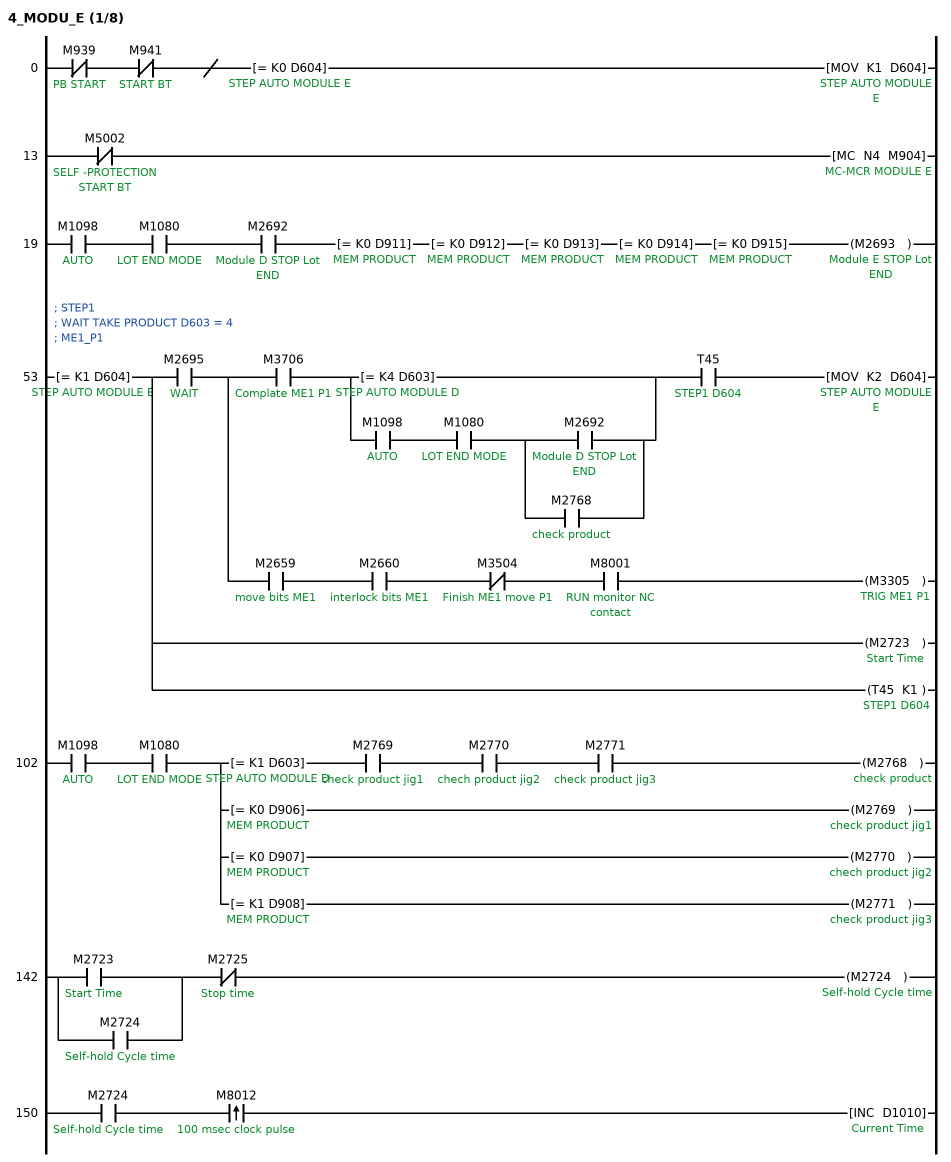
[picture p48: ladder of 4_MODU_E, rungs at steps 0 to 150]
0     LDI     M939  ; PB START
      ANI     M941  ; START BT
      INV
      AND=    K0 D604  ; STEP AUTO MODULE E
      MOV     K1 D604
13    LDI     M5002  ; SELF -PROTECTION START BT
      MC      N4 M904  ; MC-MCR MODULE E
19    LD      M1098  ; AUTO
      AND     M1080  ; LOT END MODE
      AND     M2692  ; Module D STOP Lot END
      AND=    K0 D911  ; MEM PRODUCT
      AND=    K0 D912  ; MEM PRODUCT
      AND=    K0 D913  ; MEM PRODUCT
      AND=    K0 D914  ; MEM PRODUCT
      AND=    K0 D915  ; MEM PRODUCT
      OUT     M2693  ; Module E STOP Lot END
; STEP1
; WAIT TAKE PRODUCT D603 = 4
; ME1_P1
53    LD=     K1 D604  ; STEP AUTO MODULE E
      MPS
      AND     M2695  ; WAIT
      MPS
      AND     M3706  ; Complate ME1 P1
      LD=     K4 D603  ; STEP AUTO MODULE D
      LD      M1098  ; AUTO
      AND     M1080  ; LOT END MODE
      LD      M2692  ; Module D STOP Lot END
      OR      M2768  ; check product
      ANB
      ORB
      ANB
      AND     T45  ; STEP1 D604
      MOV     K2 D604
      MPP
      AND     M2659  ; move bits ME1
      AND     M2660  ; interlock bits ME1
      ANI     M3504  ; Finish ME1 move P1
      AND     M8001  ; RUN monitor NC contact
      OUT     M3305  ; TRIG ME1 P1
        [note] TRIG ME1 P1
      MPP
      OUT     M2723  ; Start Time
      OUT     T45 K1  ; STEP1 D604
102   LD      M1098  ; AUTO
      AND     M1080  ; LOT END MODE
      MPS
      AND=    K1 D603  ; STEP AUTO MODULE D
      AND     M2769  ; check product jig1
      AND     M2770  ; chech product jig2
      AND     M2771  ; check product jig3
      OUT     M2768  ; check product
      MRD
      AND=    K0 D906  ; MEM PRODUCT
      OUT     M2769  ; check product jig1
      MRD
      AND=    K0 D907  ; MEM PRODUCT
      OUT     M2770  ; chech product jig2
      MPP
      AND=    K1 D908  ; MEM PRODUCT
      OUT     M2771  ; check product jig3
142   LD      M2723  ; Start Time
      OR      M2724  ; Self-hold Cycle time
      ANI     M2725  ; Stop time
      OUT     M2724  ; Self-hold Cycle time
150   LD      M2724  ; Self-hold Cycle time
      ANDP    M8012  ; 100 msec clock pulse
      INC     D1010  ; Current Time
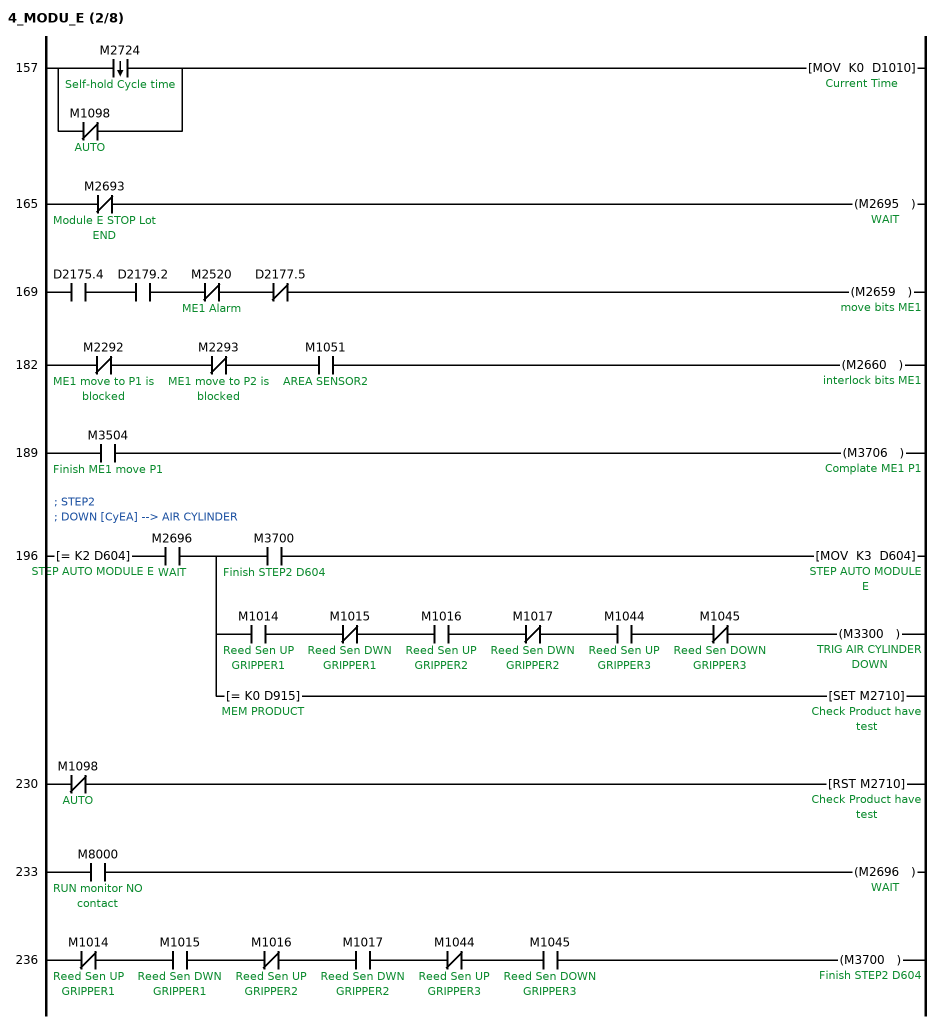
157   LDF     M2724  ; Self-hold Cycle time
      ORI     M1098  ; AUTO
      MOV     K0 D1010
165   LDI     M2693  ; Module E STOP Lot END
      OUT     M2695  ; WAIT
169   LD      D2175.4
      AND     D2179.2
      ANI     M2520  ; ME1 Alarm
      ANI     D2177.5
      OUT     M2659  ; move bits ME1
182   LDI     M2292  ; ME1 move to P1 is blocked
      ANI     M2293  ; ME1 move to P2 is blocked
      AND     M1051  ; AREA SENSOR2
      OUT     M2660  ; interlock bits ME1
189   LD      M3504  ; Finish ME1 move P1
      OUT     M3706  ; Complate ME1 P1
; STEP2
; DOWN [CyEA] --> AIR CYLINDER
196   LD=     K2 D604  ; STEP AUTO MODULE E
      AND     M2696  ; WAIT
      MPS
      AND     M3700  ; Finish STEP2 D604
      MOV     K3 D604
      MRD
      AND     M1014  ; Reed Sen UP GRIPPER1
      ANI     M1015  ; Reed Sen DWN GRIPPER1
      AND     M1016  ; Reed Sen UP GRIPPER2
      ANI     M1017  ; Reed Sen DWN GRIPPER2
      AND     M1044  ; Reed Sen UP GRIPPER3
      ANI     M1045  ; Reed Sen DOWN GRIPPER3
      OUT     M3300  ; TRIG AIR CYLINDER DOWN
        [note] TRIG AIR CYLINDER DOWN
      MPP
      AND=    K0 D915  ; MEM PRODUCT
      SET     M2710  ; Check Product have test
230   LDI     M1098  ; AUTO
      RST     M2710  ; Check Product have test
233   LD      M8000  ; RUN monitor NO contact
      OUT     M2696  ; WAIT
236   LDI     M1014  ; Reed Sen UP GRIPPER1
      AND     M1015  ; Reed Sen DWN GRIPPER1
      ANI     M1016  ; Reed Sen UP GRIPPER2
      AND     M1017  ; Reed Sen DWN GRIPPER2
      ANI     M1044  ; Reed Sen UP GRIPPER3
      AND     M1045  ; Reed Sen DOWN GRIPPER3
      OUT     M3700  ; Finish STEP2 D604
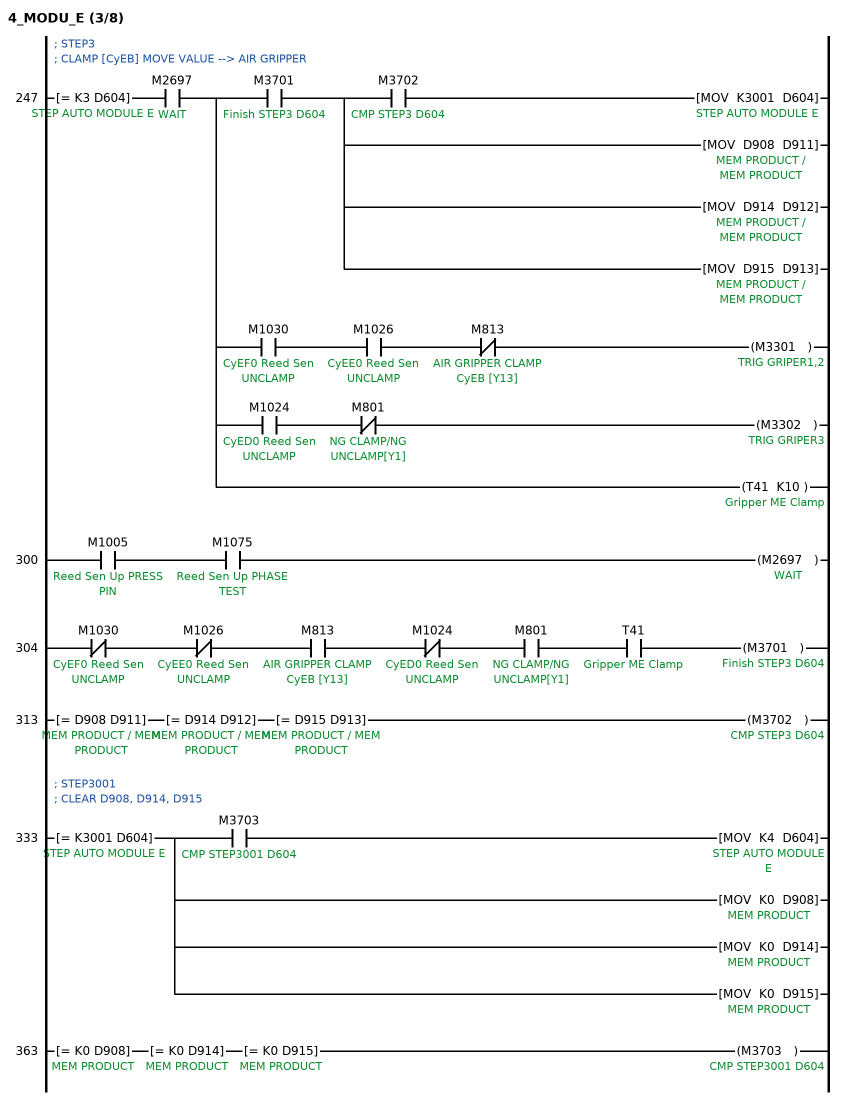
; STEP3
; CLAMP [CyEB] MOVE VALUE --> AIR GRIPPER
247   LD=     K3 D604  ; STEP AUTO MODULE E
      AND     M2697  ; WAIT
      MPS
      AND     M3701  ; Finish STEP3 D604
      MPS
      AND     M3702  ; CMP STEP3 D604
      MOV     K3001 D604
      MPP
      MOV     D908 D911
      MOV     D914 D912
      MOV     D915 D913
      MRD
      AND     M1030  ; CyEF0 Reed Sen UNCLAMP
      AND     M1026  ; CyEE0 Reed Sen UNCLAMP
      ANI     M813  ; AIR GRIPPER CLAMP CyEB [Y13]
      OUT     M3301  ; TRIG GRIPER1,2
        [note] TRIG GRIPER1,2
      MRD
      AND     M1024  ; CyED0 Reed Sen UNCLAMP
      ANI     M801  ; NG CLAMP/NG UNCLAMP[Y1]
      OUT     M3302  ; TRIG GRIPER3
        [note] TRIG GRIPER3
      MPP
      OUT     T41 K10  ; Gripper ME Clamp
300   LD      M1005  ; Reed Sen Up PRESS PIN
      AND     M1075  ; Reed Sen Up PHASE TEST
      OUT     M2697  ; WAIT
304   LDI     M1030  ; CyEF0 Reed Sen UNCLAMP
      ANI     M1026  ; CyEE0 Reed Sen UNCLAMP
      AND     M813  ; AIR GRIPPER CLAMP CyEB [Y13]
      ANI     M1024  ; CyED0 Reed Sen UNCLAMP
      AND     M801  ; NG CLAMP/NG UNCLAMP[Y1]
      AND     T41  ; Gripper ME Clamp
      OUT     M3701  ; Finish STEP3 D604
313   LD=     D908 D911  ; MEM PRODUCT / MEM PRODUCT
      AND=    D914 D912  ; MEM PRODUCT / MEM PRODUCT
      AND=    D915 D913  ; MEM PRODUCT / MEM PRODUCT
      OUT     M3702  ; CMP STEP3 D604
; STEP3001
; CLEAR D908, D914, D915
333   LD=     K3001 D604  ; STEP AUTO MODULE E
      MPS
      AND     M3703  ; CMP STEP3001 D604
      MOV     K4 D604
      MPP
      MOV     K0 D908
      MOV     K0 D914
      MOV     K0 D915
363   LD=     K0 D908  ; MEM PRODUCT
      AND=    K0 D914  ; MEM PRODUCT
      AND=    K0 D915  ; MEM PRODUCT
      OUT     M3703  ; CMP STEP3001 D604
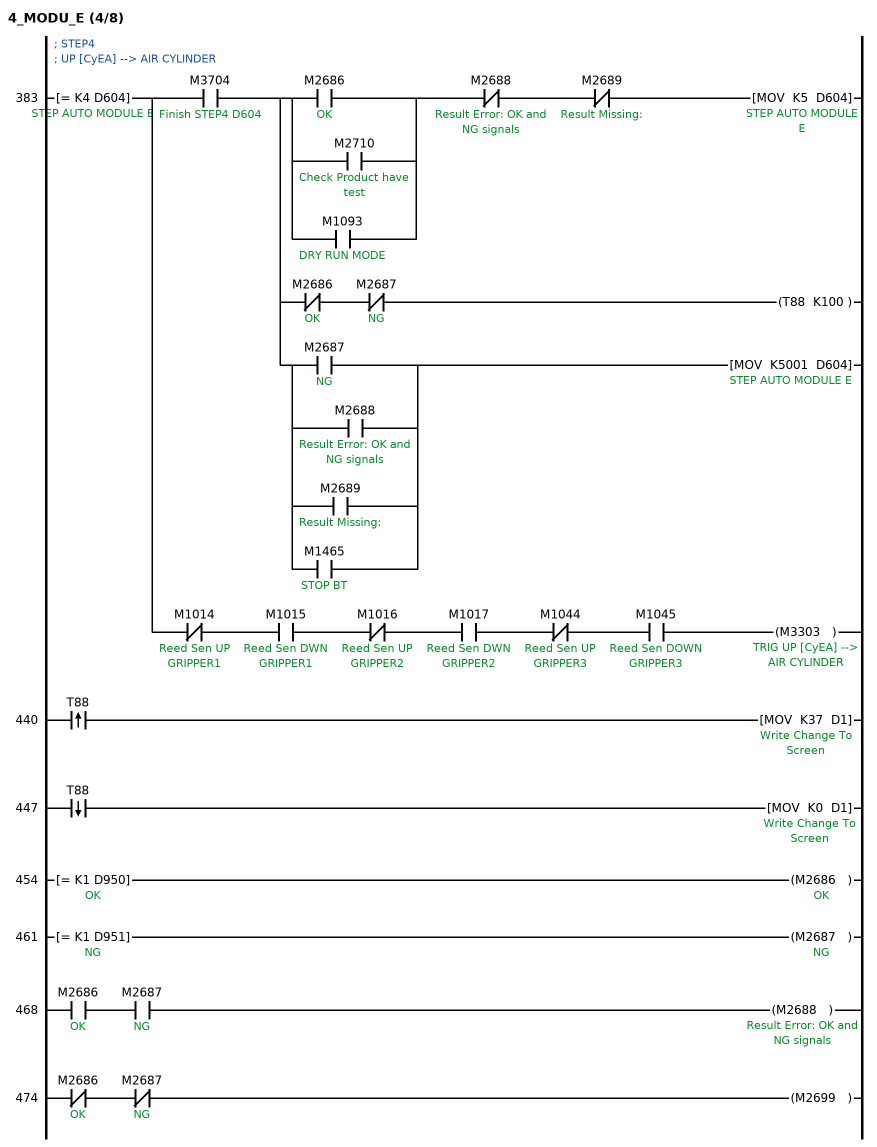
; STEP4
; UP [CyEA] --> AIR CYLINDER
383   LD=     K4 D604  ; STEP AUTO MODULE E
      MPS
      AND     M3704  ; Finish STEP4 D604
      MPS
      LD      M2686  ; OK
      OR      M2710  ; Check Product have test
      OR      M1093  ; DRY RUN MODE
      ANB
      ANI     M2688  ; Result Error: OK and NG signals
      ANI     M2689  ; Result Missing:
      MOV     K5 D604
      MRD
      ANI     M2686  ; OK
      ANI     M2687  ; NG
      OUT     T88 K100
      MPP
      LD      M2687  ; NG
      OR      M2688  ; Result Error: OK and NG signals
      OR      M2689  ; Result Missing:
      OR      M1465  ; STOP BT
      ANB
      MOV     K5001 D604
      MPP
      ANI     M1014  ; Reed Sen UP GRIPPER1
      AND     M1015  ; Reed Sen DWN GRIPPER1
      ANI     M1016  ; Reed Sen UP GRIPPER2
      AND     M1017  ; Reed Sen DWN GRIPPER2
      ANI     M1044  ; Reed Sen UP GRIPPER3
      AND     M1045  ; Reed Sen DOWN GRIPPER3
      OUT     M3303  ; TRIG UP [CyEA] --> AIR CYLINDER
        [note] TRIG UP AIR CYLINDER
440   LDP     T88
      MOV     K37 D1  ; Write Change To Screen
447   LDF     T88
      MOV     K0 D1
454   LD=     K1 D950  ; OK
      OUT     M2686  ; OK
461   LD=     K1 D951  ; NG
      OUT     M2687  ; NG
468   LD      M2686  ; OK
      AND     M2687  ; NG
      OUT     M2688  ; Result Error: OK and NG signals
474   LDI     M2686  ; OK
      ANI     M2687  ; NG
      OUT     M2699
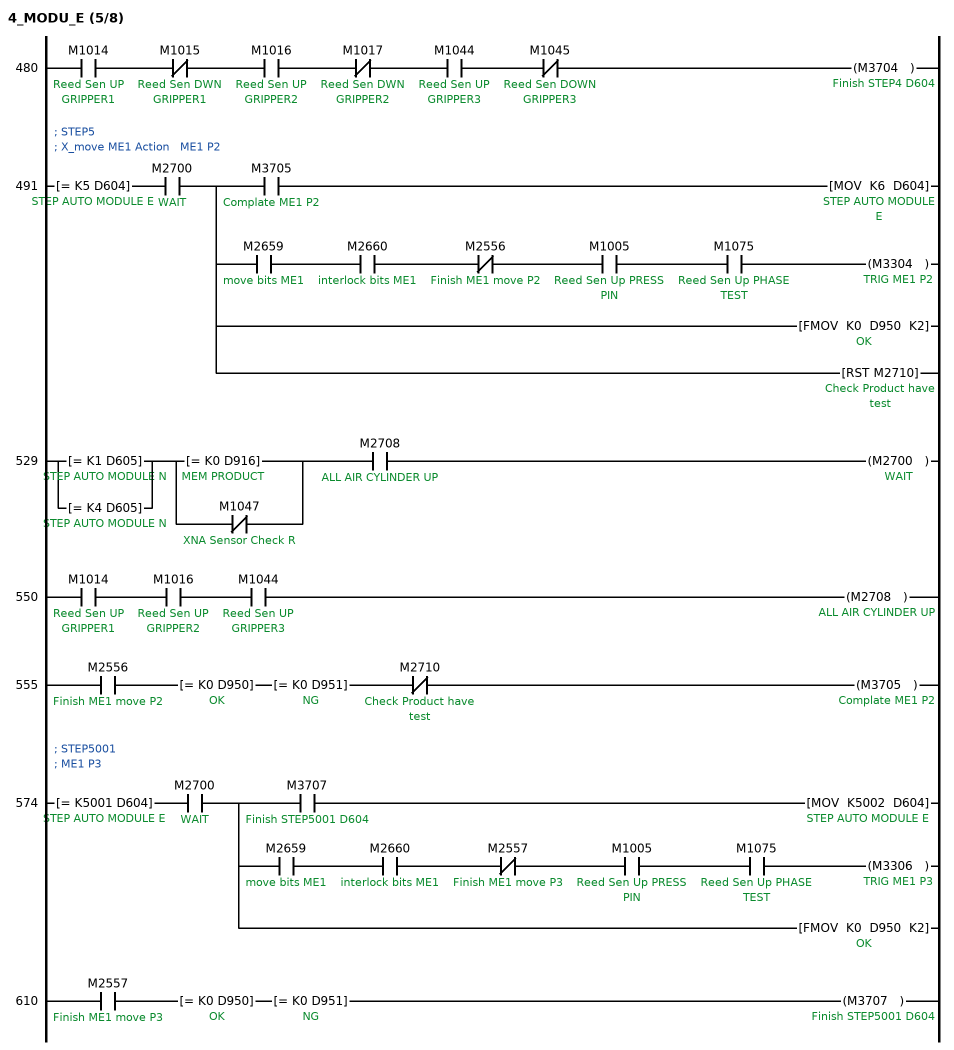
480   LD      M1014  ; Reed Sen UP GRIPPER1
      ANI     M1015  ; Reed Sen DWN GRIPPER1
      AND     M1016  ; Reed Sen UP GRIPPER2
      ANI     M1017  ; Reed Sen DWN GRIPPER2
      AND     M1044  ; Reed Sen UP GRIPPER3
      ANI     M1045  ; Reed Sen DOWN GRIPPER3
      OUT     M3704  ; Finish STEP4 D604
; STEP5
; X_move ME1 Action   ME1 P2
491   LD=     K5 D604  ; STEP AUTO MODULE E
      AND     M2700  ; WAIT
      MPS
      AND     M3705  ; Complate ME1 P2
      MOV     K6 D604
      MRD
      AND     M2659  ; move bits ME1
      AND     M2660  ; interlock bits ME1
      ANI     M2556  ; Finish ME1 move P2
      AND     M1005  ; Reed Sen Up PRESS PIN
      AND     M1075  ; Reed Sen Up PHASE TEST
      OUT     M3304  ; TRIG ME1 P2
        [note] TRIG ME1 P2
      MPP
      FMOV    K0 D950 K2
      RST     M2710  ; Check Product have test
529   LD=     K1 D605  ; STEP AUTO MODULE N
      OR=     K4 D605  ; STEP AUTO MODULE N
      LD=     K0 D916  ; MEM PRODUCT
      ORI     M1047  ; XNA Sensor Check R
      ANB
      AND     M2708  ; ALL AIR CYLINDER UP
      OUT     M2700  ; WAIT
550   LD      M1014  ; Reed Sen UP GRIPPER1
      AND     M1016  ; Reed Sen UP GRIPPER2
      AND     M1044  ; Reed Sen UP GRIPPER3
      OUT     M2708  ; ALL AIR CYLINDER UP
555   LD      M2556  ; Finish ME1 move P2
      AND=    K0 D950  ; OK
      AND=    K0 D951  ; NG
      ANI     M2710  ; Check Product have test
      OUT     M3705  ; Complate ME1 P2
; STEP5001
; ME1 P3
574   LD=     K5001 D604  ; STEP AUTO MODULE E
      AND     M2700  ; WAIT
      MPS
      AND     M3707  ; Finish STEP5001 D604
      MOV     K5002 D604
      MRD
      AND     M2659  ; move bits ME1
      AND     M2660  ; interlock bits ME1
      ANI     M2557  ; Finish ME1 move P3
      AND     M1005  ; Reed Sen Up PRESS PIN
      AND     M1075  ; Reed Sen Up PHASE TEST
      OUT     M3306  ; TRIG ME1 P3
        [note] TRIG ME1 P3
      MPP
      FMOV    K0 D950 K2
610   LD      M2557  ; Finish ME1 move P3
      AND=    K0 D950  ; OK
      AND=    K0 D951  ; NG
      OUT     M3707  ; Finish STEP5001 D604
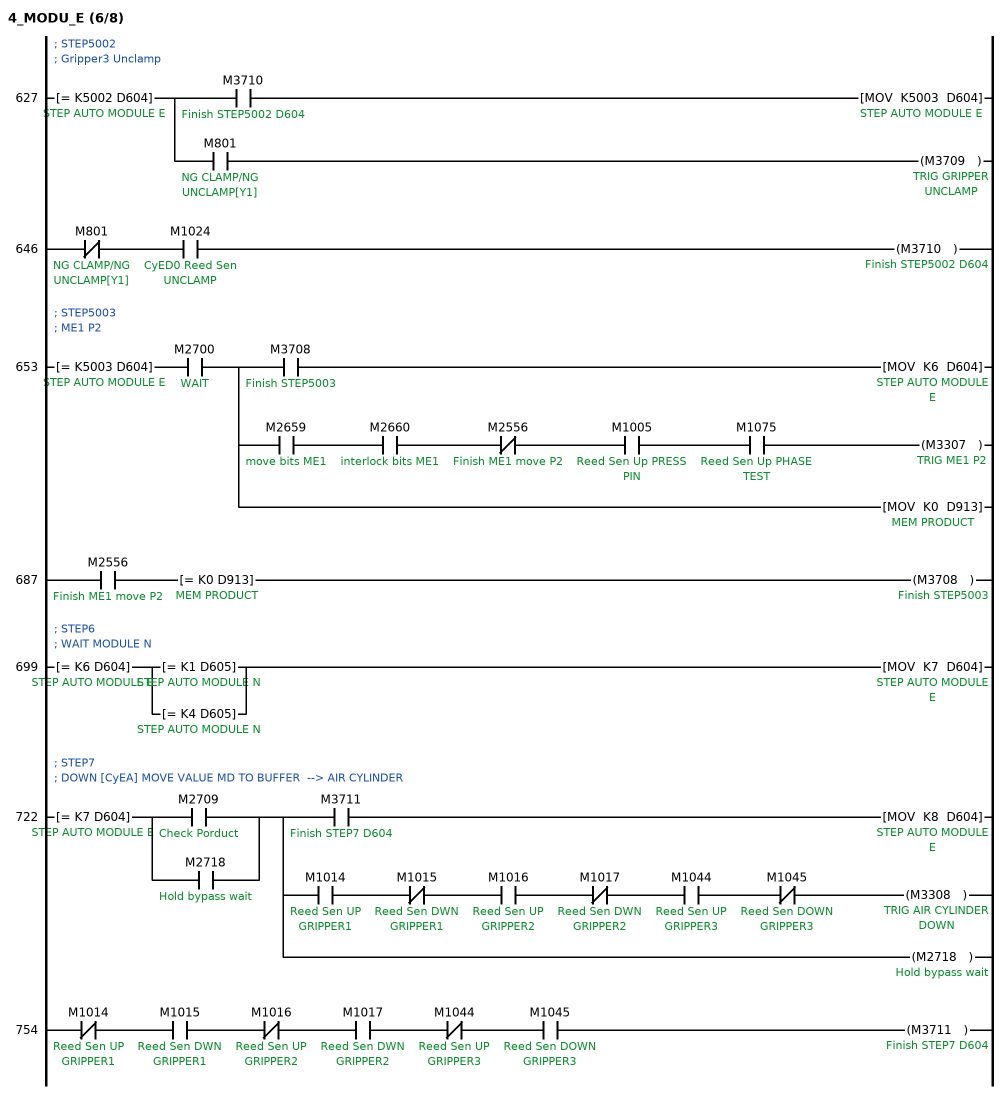
; STEP5002
; Gripper3 Unclamp
627   LD=     K5002 D604  ; STEP AUTO MODULE E
      MPS
      AND     M3710  ; Finish STEP5002 D604
      MOV     K5003 D604
      MPP
      AND     M801  ; NG CLAMP/NG UNCLAMP[Y1]
      OUT     M3709  ; TRIG GRIPPER UNCLAMP
646   LDI     M801  ; NG CLAMP/NG UNCLAMP[Y1]
      AND     M1024  ; CyED0 Reed Sen UNCLAMP
      OUT     M3710  ; Finish STEP5002 D604
; STEP5003
; ME1 P2
653   LD=     K5003 D604  ; STEP AUTO MODULE E
      AND     M2700  ; WAIT
      MPS
      AND     M3708  ; Finish STEP5003
      MOV     K6 D604
      MRD
      AND     M2659  ; move bits ME1
      AND     M2660  ; interlock bits ME1
      ANI     M2556  ; Finish ME1 move P2
      AND     M1005  ; Reed Sen Up PRESS PIN
      AND     M1075  ; Reed Sen Up PHASE TEST
      OUT     M3307  ; TRIG ME1 P2
        [note] TRIG ME1 P2
      MPP
      MOV     K0 D913
687   LD      M2556  ; Finish ME1 move P2
      AND=    K0 D913  ; MEM PRODUCT
      OUT     M3708  ; Finish STEP5003
; STEP6
; WAIT MODULE N
699   LD=     K6 D604  ; STEP AUTO MODULE E
      LD=     K1 D605  ; STEP AUTO MODULE N
      OR=     K4 D605  ; STEP AUTO MODULE N
      ANB
      MOV     K7 D604
; STEP7
; DOWN [CyEA] MOVE VALUE MD TO BUFFER  --> AIR CYLINDER
722   LD=     K7 D604  ; STEP AUTO MODULE E
      LD      M2709  ; Check Porduct
      OR      M2718  ; Hold bypass wait
      ANB
      MPS
      AND     M3711  ; Finish STEP7 D604
      MOV     K8 D604
      MRD
      AND     M1014  ; Reed Sen UP GRIPPER1
      ANI     M1015  ; Reed Sen DWN GRIPPER1
      AND     M1016  ; Reed Sen UP GRIPPER2
      ANI     M1017  ; Reed Sen DWN GRIPPER2
      AND     M1044  ; Reed Sen UP GRIPPER3
      ANI     M1045  ; Reed Sen DOWN GRIPPER3
      OUT     M3308  ; TRIG AIR CYLINDER DOWN
        [note] TRIG AIR CYLINDER DOWN
      MPP
      OUT     M2718  ; Hold bypass wait
754   LDI     M1014  ; Reed Sen UP GRIPPER1
      AND     M1015  ; Reed Sen DWN GRIPPER1
      ANI     M1016  ; Reed Sen UP GRIPPER2
      AND     M1017  ; Reed Sen DWN GRIPPER2
      ANI     M1044  ; Reed Sen UP GRIPPER3
      AND     M1045  ; Reed Sen DOWN GRIPPER3
      OUT     M3711  ; Finish STEP7 D604
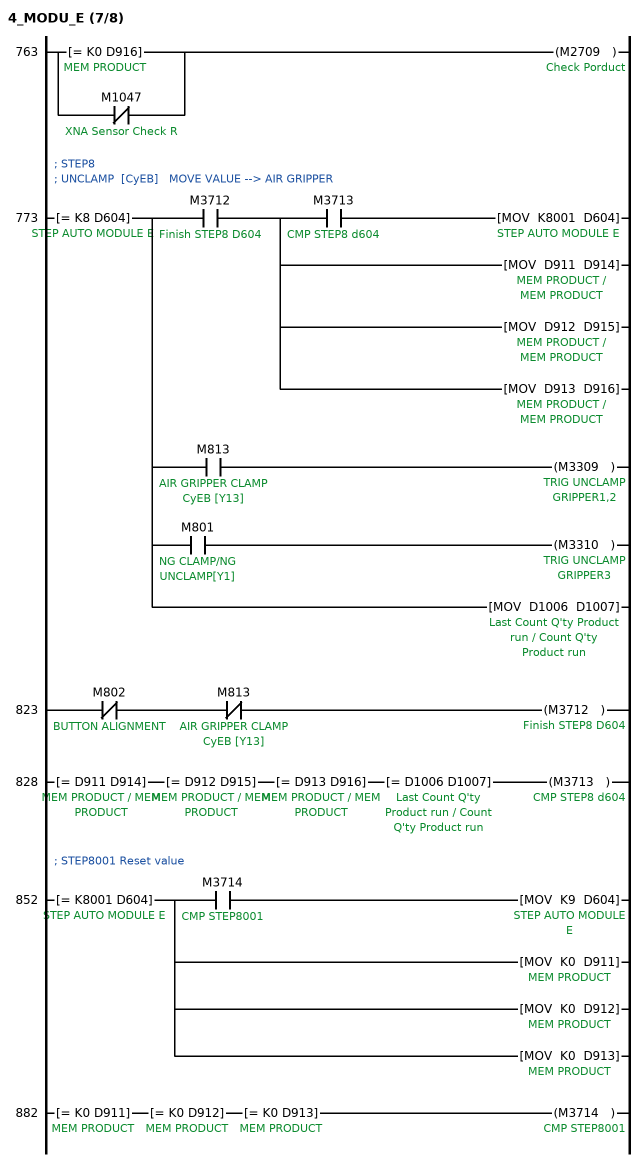
763   LD=     K0 D916  ; MEM PRODUCT
      ORI     M1047  ; XNA Sensor Check R
      OUT     M2709  ; Check Porduct
; STEP8
; UNCLAMP  [CyEB]   MOVE VALUE --> AIR GRIPPER
773   LD=     K8 D604  ; STEP AUTO MODULE E
      MPS
      AND     M3712  ; Finish STEP8 D604
      MPS
      AND     M3713  ; CMP STEP8 d604
      MOV     K8001 D604
      MPP
      MOV     D911 D914
      MOV     D912 D915
      MOV     D913 D916
      MRD
      AND     M813  ; AIR GRIPPER CLAMP CyEB [Y13]
      OUT     M3309  ; TRIG UNCLAMP GRIPPER1,2
        [note] TRIG UNCLAMP GRIPPER1,2
      MRD
      AND     M801  ; NG CLAMP/NG UNCLAMP[Y1]
      OUT     M3310  ; TRIG UNCLAMP GRIPPER3
        [note] TRIG UNCLAMP GRIPPER3
      MPP
      MOV     D1006 D1007  ; Last Count Q'ty Product run / Count Q'ty Product run
823   LDI     M802  ; BUTTON ALIGNMENT
      ANI     M813  ; AIR GRIPPER CLAMP CyEB [Y13]
      OUT     M3712  ; Finish STEP8 D604
828   LD=     D911 D914  ; MEM PRODUCT / MEM PRODUCT
      AND=    D912 D915  ; MEM PRODUCT / MEM PRODUCT
      AND=    D913 D916  ; MEM PRODUCT / MEM PRODUCT
      AND=    D1006 D1007  ; Last Count Q'ty Product run / Count Q'ty Product run
      OUT     M3713  ; CMP STEP8 d604
; STEP8001 Reset value
852   LD=     K8001 D604  ; STEP AUTO MODULE E
      MPS
      AND     M3714  ; CMP STEP8001
      MOV     K9 D604
      MPP
      MOV     K0 D911
      MOV     K0 D912
      MOV     K0 D913
882   LD=     K0 D911  ; MEM PRODUCT
      AND=    K0 D912  ; MEM PRODUCT
      AND=    K0 D913  ; MEM PRODUCT
      OUT     M3714  ; CMP STEP8001
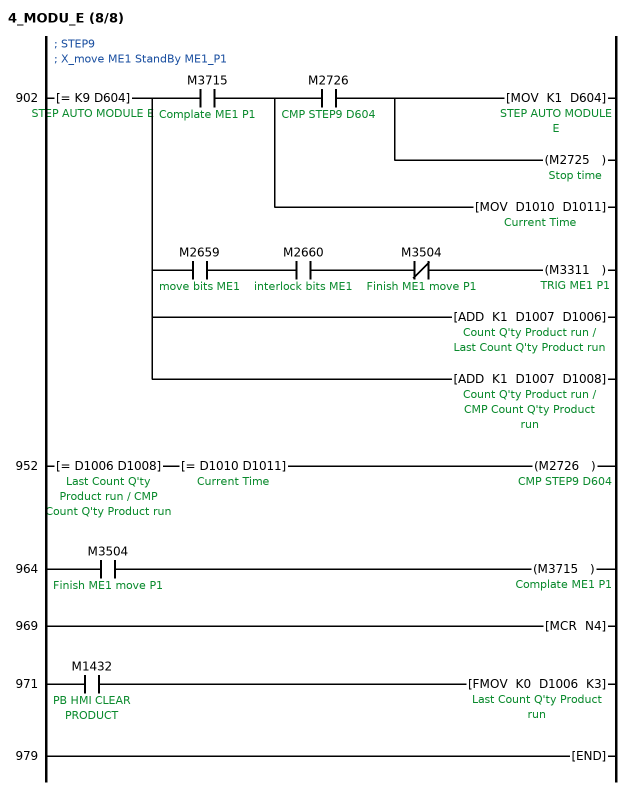
; STEP9
; X_move ME1 StandBy ME1_P1
902   LD=     K9 D604  ; STEP AUTO MODULE E
      MPS
      AND     M3715  ; Complate ME1 P1
      MPS
      AND     M2726  ; CMP STEP9 D604
      MOV     K1 D604
      OUT     M2725  ; Stop time
      MPP
      MOV     D1010 D1011
      MRD
      AND     M2659  ; move bits ME1
      AND     M2660  ; interlock bits ME1
      ANI     M3504  ; Finish ME1 move P1
      OUT     M3311  ; TRIG ME1 P1
        [note] TRIG ME1 P1
      MPP
      ADD     K1 D1007 D1006
      ADD     K1 D1007 D1008  ; CMP Count Q'ty Product run
952   LD=     D1006 D1008  ; Last Count Q'ty Product run / CMP Count Q'ty Product run
      AND=    D1010 D1011  ; Current Time
      OUT     M2726  ; CMP STEP9 D604
964   LD      M3504  ; Finish ME1 move P1
      OUT     M3715  ; Complate ME1 P1
969   MCR     N4
971   LD      M1432  ; PB HMI CLEAR PRODUCT
      FMOV    K0 D1006 K3
979   END
END_PROGRAM

PROGRAM 5_MODU_N
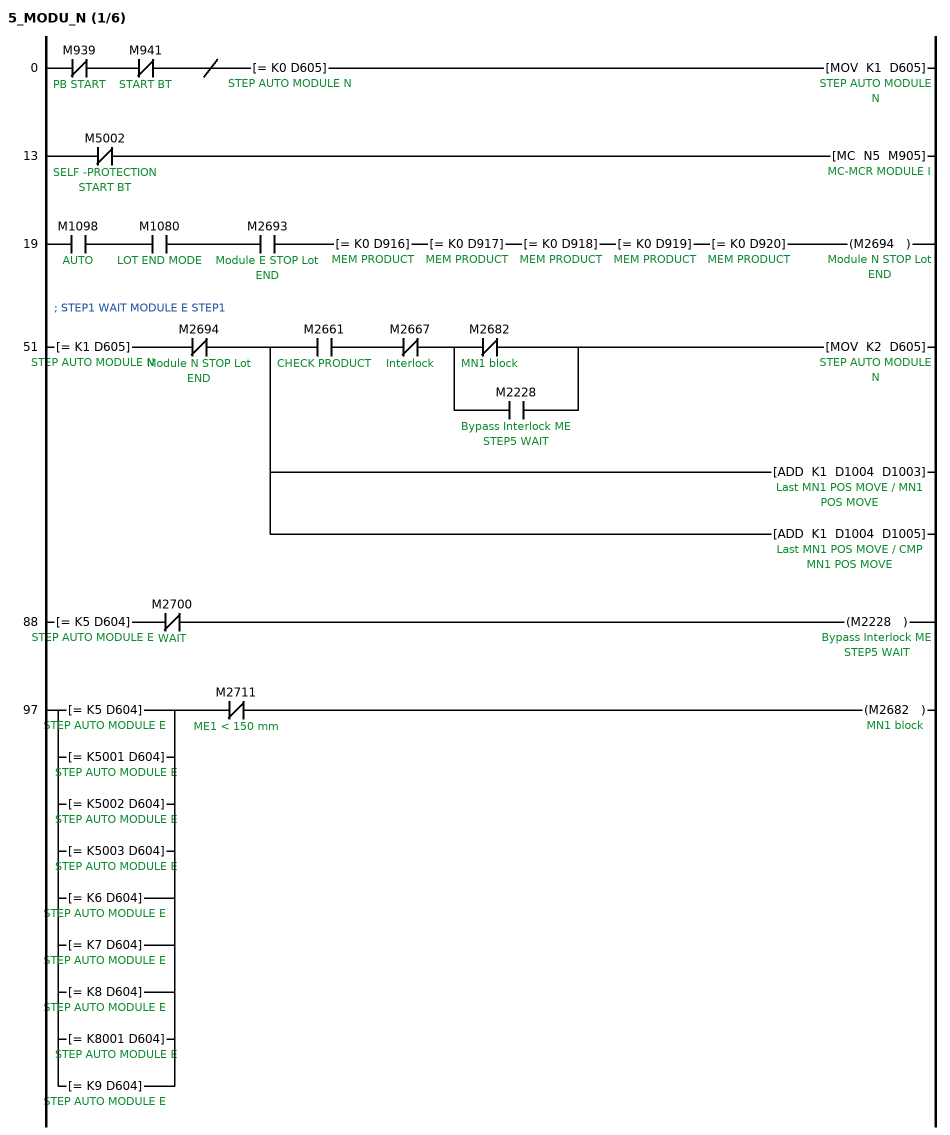
0     LDI     M939  ; PB START
      ANI     M941  ; START BT
      INV
      AND=    K0 D605  ; STEP AUTO MODULE N
      MOV     K1 D605
13    LDI     M5002  ; SELF -PROTECTION START BT
      MC      N5 M905  ; MC-MCR MODULE I
19    LD      M1098  ; AUTO
      AND     M1080  ; LOT END MODE
      AND     M2693  ; Module E STOP Lot END
      AND=    K0 D916  ; MEM PRODUCT
      AND=    K0 D917  ; MEM PRODUCT
      AND=    K0 D918  ; MEM PRODUCT
      AND=    K0 D919  ; MEM PRODUCT
      AND=    K0 D920  ; MEM PRODUCT
      OUT     M2694  ; Module N STOP Lot END
; STEP1 WAIT MODULE E STEP1
51    LD=     K1 D605  ; STEP AUTO MODULE N
      ANI     M2694  ; Module N STOP Lot END
      MPS
      AND     M2661  ; CHECK PRODUCT
      ANI     M2667  ; Interlock
      LDI     M2682  ; MN1 block
      OR      M2228  ; Bypass Interlock ME STEP5 WAIT
      ANB
      MOV     K2 D605
      MPP
      ADD     K1 D1004 D1003  ; Last MN1 POS MOVE / MN1 POS MOVE
      ADD     K1 D1004 D1005  ; CMP MN1 POS MOVE
88    LD=     K5 D604  ; STEP AUTO MODULE E
      ANI     M2700  ; WAIT
      OUT     M2228  ; Bypass Interlock ME STEP5 WAIT
97    LD=     K5 D604  ; STEP AUTO MODULE E
      OR=     K5001 D604  ; STEP AUTO MODULE E
      OR=     K5002 D604  ; STEP AUTO MODULE E
      OR=     K5003 D604  ; STEP AUTO MODULE E
      OR=     K6 D604  ; STEP AUTO MODULE E
      OR=     K7 D604  ; STEP AUTO MODULE E
      OR=     K8 D604  ; STEP AUTO MODULE E
      OR=     K8001 D604  ; STEP AUTO MODULE E
      OR=     K9 D604  ; STEP AUTO MODULE E
      ANI     M2711  ; ME1 < 150 mm
      OUT     M2682  ; MN1 block
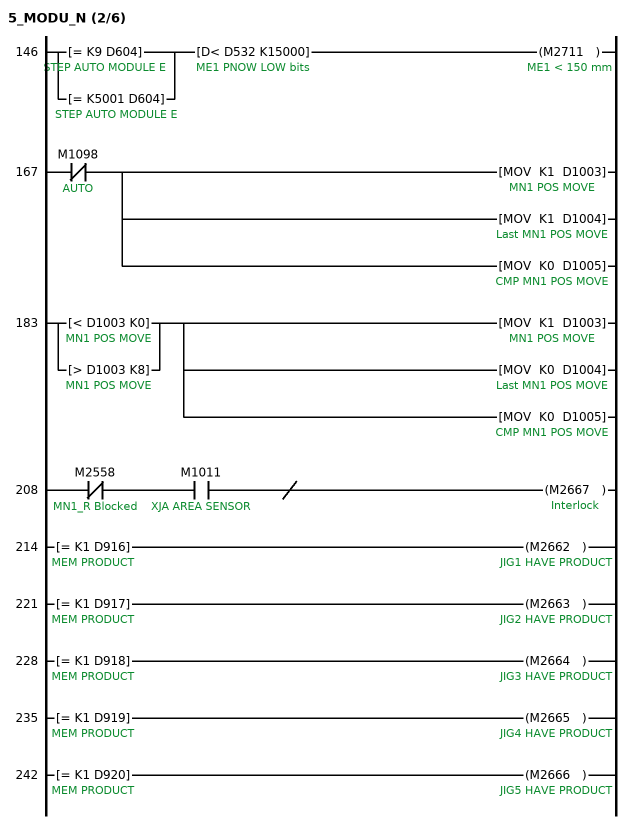
146   LD=     K9 D604  ; STEP AUTO MODULE E
      OR=     K5001 D604  ; STEP AUTO MODULE E
      ANDD<   D532 K15000  ; ME1 PNOW LOW bits
      OUT     M2711  ; ME1 < 150 mm
167   LDI     M1098  ; AUTO
      MOV     K1 D1003
      MOV     K1 D1004
      MOV     K0 D1005
183   LD<     D1003 K0  ; MN1 POS MOVE
      OR>     D1003 K8  ; MN1 POS MOVE
      MOV     K1 D1003
      MOV     K0 D1004
      MOV     K0 D1005
208   LDI     M2558  ; MN1_R Blocked
      AND     M1011  ; XJA AREA SENSOR
      INV
      OUT     M2667  ; Interlock
214   LD=     K1 D916  ; MEM PRODUCT
      OUT     M2662  ; JIG1 HAVE PRODUCT
221   LD=     K1 D917  ; MEM PRODUCT
      OUT     M2663  ; JIG2 HAVE PRODUCT
228   LD=     K1 D918  ; MEM PRODUCT
      OUT     M2664  ; JIG3 HAVE PRODUCT
235   LD=     K1 D919  ; MEM PRODUCT
      OUT     M2665  ; JIG4 HAVE PRODUCT
242   LD=     K1 D920  ; MEM PRODUCT
      OUT     M2666  ; JIG5 HAVE PRODUCT
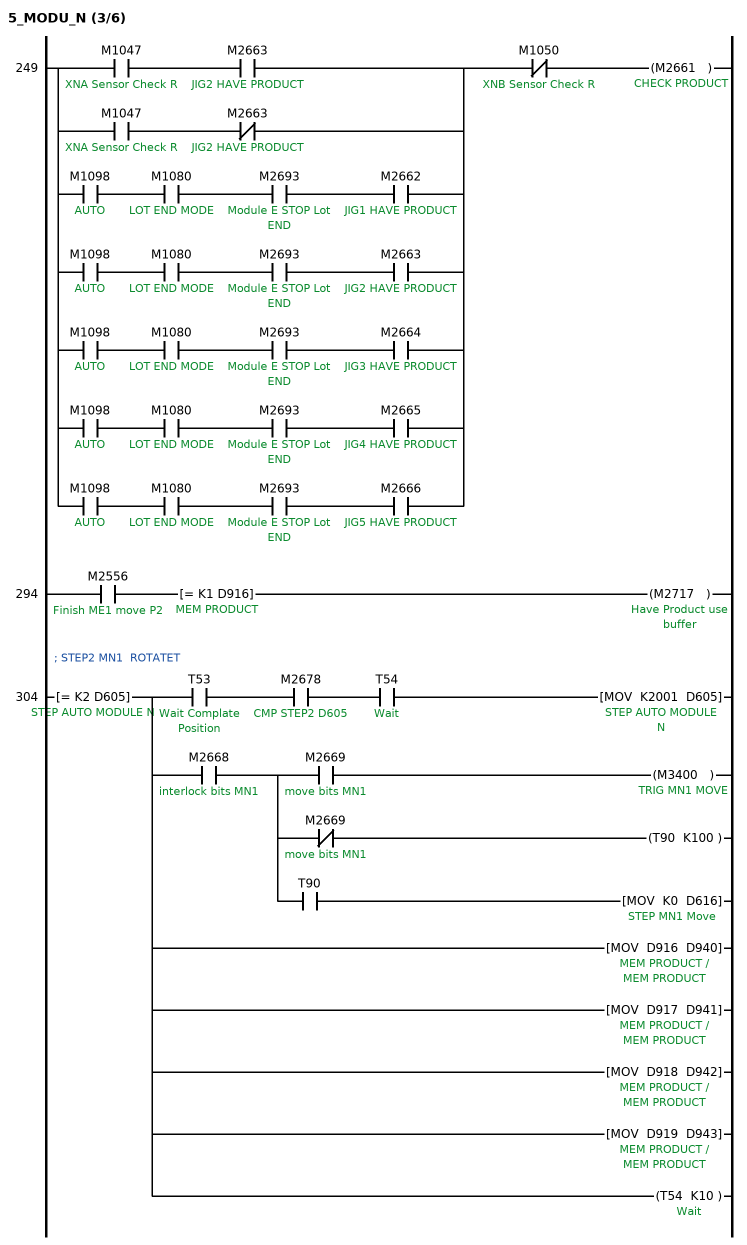
249   LD      M1047  ; XNA Sensor Check R
      AND     M2663  ; JIG2 HAVE PRODUCT
      LD      M1047  ; XNA Sensor Check R
      ANI     M2663  ; JIG2 HAVE PRODUCT
      ORB
      LD      M1098  ; AUTO
      AND     M1080  ; LOT END MODE
      AND     M2693  ; Module E STOP Lot END
      AND     M2662  ; JIG1 HAVE PRODUCT
      ORB
      LD      M1098  ; AUTO
      AND     M1080  ; LOT END MODE
      AND     M2693  ; Module E STOP Lot END
      AND     M2663  ; JIG2 HAVE PRODUCT
      ORB
      LD      M1098  ; AUTO
      AND     M1080  ; LOT END MODE
      AND     M2693  ; Module E STOP Lot END
      AND     M2664  ; JIG3 HAVE PRODUCT
      ORB
      LD      M1098  ; AUTO
      AND     M1080  ; LOT END MODE
      AND     M2693  ; Module E STOP Lot END
      AND     M2665  ; JIG4 HAVE PRODUCT
      ORB
      LD      M1098  ; AUTO
      AND     M1080  ; LOT END MODE
      AND     M2693  ; Module E STOP Lot END
      AND     M2666  ; JIG5 HAVE PRODUCT
      ORB
      ANI     M1050  ; XNB Sensor Check R
      OUT     M2661  ; CHECK PRODUCT
294   LD      M2556  ; Finish ME1 move P2
      AND=    K1 D916  ; MEM PRODUCT
      OUT     M2717  ; Have Product use buffer
; STEP2 MN1  ROTATET
304   LD=     K2 D605  ; STEP AUTO MODULE N
      MPS
      AND     T53  ; Wait Complate Position
      AND     M2678  ; CMP STEP2 D605
      AND     T54  ; Wait
      MOV     K2001 D605
      MRD
      AND     M2668  ; interlock bits MN1
      MPS
      AND     M2669  ; move bits MN1
      OUT     M3400  ; TRIG MN1 MOVE
        [note] TRIG MD1 MOVE
      MRD
      ANI     M2669  ; move bits MN1
      OUT     T90 K100
      MPP
      AND     T90
      MOV     K0 D616  ; STEP MN1 Move
      MPP
      MOV     D916 D940  ; MEM PRODUCT
      MOV     D917 D941  ; MEM PRODUCT
      MOV     D918 D942  ; MEM PRODUCT
      MOV     D919 D943  ; MEM PRODUCT
      OUT     T54 K10  ; Wait
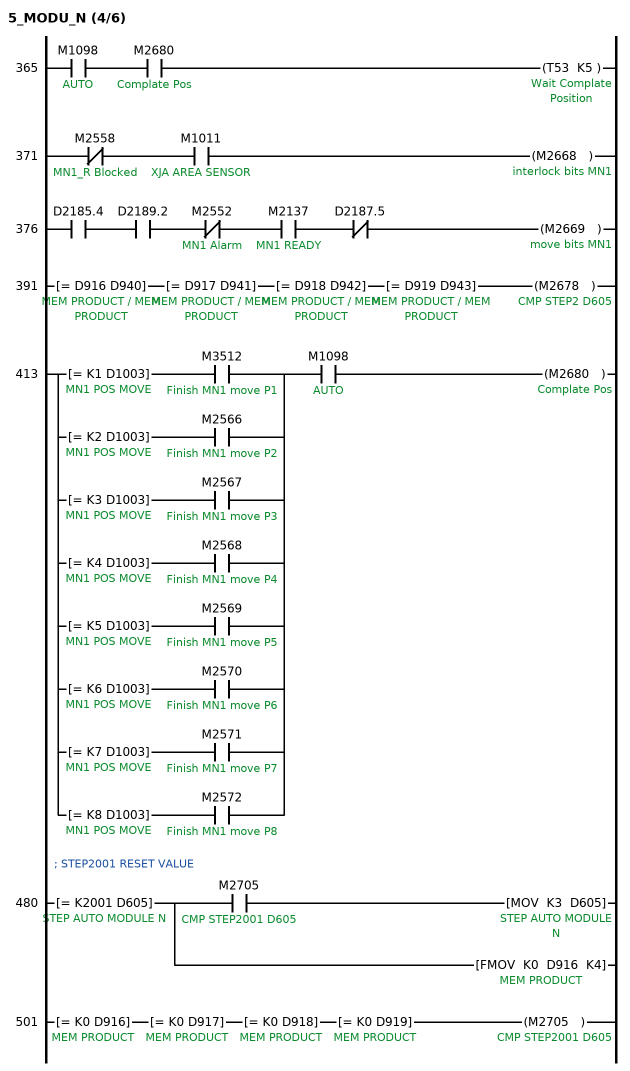
365   LD      M1098  ; AUTO
      AND     M2680  ; Complate Pos
      OUT     T53 K5  ; Wait Complate Position
371   LDI     M2558  ; MN1_R Blocked
      AND     M1011  ; XJA AREA SENSOR
      OUT     M2668  ; interlock bits MN1
376   LD      D2185.4
      AND     D2189.2
      ANI     M2552  ; MN1 Alarm
      AND     M2137  ; MN1 READY
      ANI     D2187.5
      OUT     M2669  ; move bits MN1
391   LD=     D916 D940  ; MEM PRODUCT / MEM PRODUCT
      AND=    D917 D941  ; MEM PRODUCT / MEM PRODUCT
      AND=    D918 D942  ; MEM PRODUCT / MEM PRODUCT
      AND=    D919 D943  ; MEM PRODUCT / MEM PRODUCT
      OUT     M2678  ; CMP STEP2 D605
413   LD=     K1 D1003  ; MN1 POS MOVE
      AND     M3512  ; Finish MN1 move P1
      LD=     K2 D1003  ; MN1 POS MOVE
      AND     M2566  ; Finish MN1 move P2
      ORB
      LD=     K3 D1003  ; MN1 POS MOVE
      AND     M2567  ; Finish MN1 move P3
      ORB
      LD=     K4 D1003  ; MN1 POS MOVE
      AND     M2568  ; Finish MN1 move P4
      ORB
      LD=     K5 D1003  ; MN1 POS MOVE
      AND     M2569  ; Finish MN1 move P5
      ORB
      LD=     K6 D1003  ; MN1 POS MOVE
      AND     M2570  ; Finish MN1 move P6
      ORB
      LD=     K7 D1003  ; MN1 POS MOVE
      AND     M2571  ; Finish MN1 move P7
      ORB
      LD=     K8 D1003  ; MN1 POS MOVE
      AND     M2572  ; Finish MN1 move P8
      ORB
      AND     M1098  ; AUTO
      OUT     M2680  ; Complate Pos
; STEP2001 RESET VALUE
480   LD=     K2001 D605  ; STEP AUTO MODULE N
      MPS
      AND     M2705  ; CMP STEP2001 D605
      MOV     K3 D605
      MPP
      FMOV    K0 D916 K4
501   LD=     K0 D916  ; MEM PRODUCT
      AND=    K0 D917  ; MEM PRODUCT
      AND=    K0 D918  ; MEM PRODUCT
      AND=    K0 D919  ; MEM PRODUCT
      OUT     M2705  ; CMP STEP2001 D605
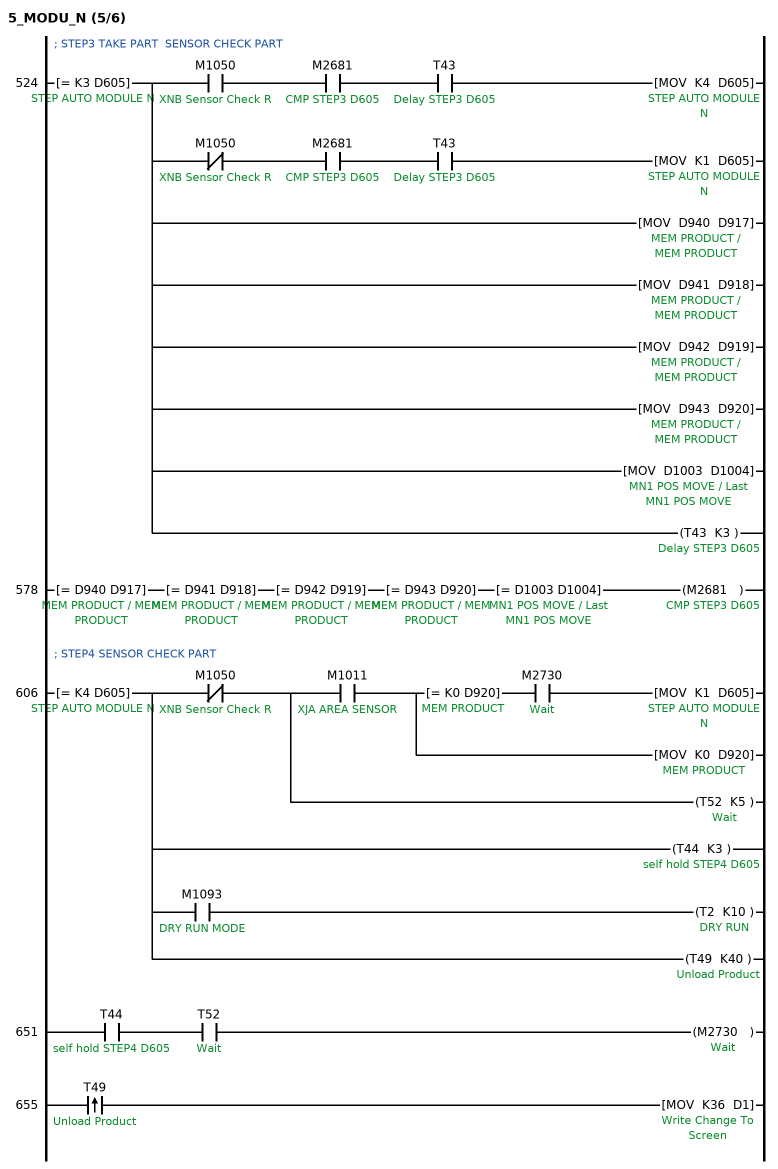
; STEP3 TAKE PART  SENSOR CHECK PART
524   LD=     K3 D605  ; STEP AUTO MODULE N
      MPS
      AND     M1050  ; XNB Sensor Check R
      AND     M2681  ; CMP STEP3 D605
      AND     T43  ; Delay STEP3 D605
      MOV     K4 D605
      MRD
      ANI     M1050  ; XNB Sensor Check R
      AND     M2681  ; CMP STEP3 D605
      AND     T43  ; Delay STEP3 D605
      MOV     K1 D605
      MPP
      MOV     D940 D917
      MOV     D941 D918
      MOV     D942 D919
      MOV     D943 D920
      MOV     D1003 D1004
      OUT     T43 K3  ; Delay STEP3 D605
578   LD=     D940 D917  ; MEM PRODUCT / MEM PRODUCT
      AND=    D941 D918  ; MEM PRODUCT / MEM PRODUCT
      AND=    D942 D919  ; MEM PRODUCT / MEM PRODUCT
      AND=    D943 D920  ; MEM PRODUCT / MEM PRODUCT
      AND=    D1003 D1004  ; MN1 POS MOVE / Last MN1 POS MOVE
      OUT     M2681  ; CMP STEP3 D605
; STEP4 SENSOR CHECK PART
606   LD=     K4 D605  ; STEP AUTO MODULE N
      MPS
      ANI     M1050  ; XNB Sensor Check R
      MPS
      AND     M1011  ; XJA AREA SENSOR
      MPS
      AND=    K0 D920  ; MEM PRODUCT
      AND     M2730  ; Wait
      MOV     K1 D605
      MPP
      MOV     K0 D920
      MPP
      OUT     T52 K5  ; Wait
      MPP
      OUT     T44 K3  ; self hold STEP4 D605
      MPS
      AND     M1093  ; DRY RUN MODE
      OUT     T2 K10  ; DRY RUN
      MPP
      OUT     T49 K40  ; Unload Product
651   LD      T44  ; self hold STEP4 D605
      AND     T52  ; Wait
      OUT     M2730  ; Wait
655   LDP     T49  ; Unload Product
      MOV     K36 D1  ; Write Change To Screen
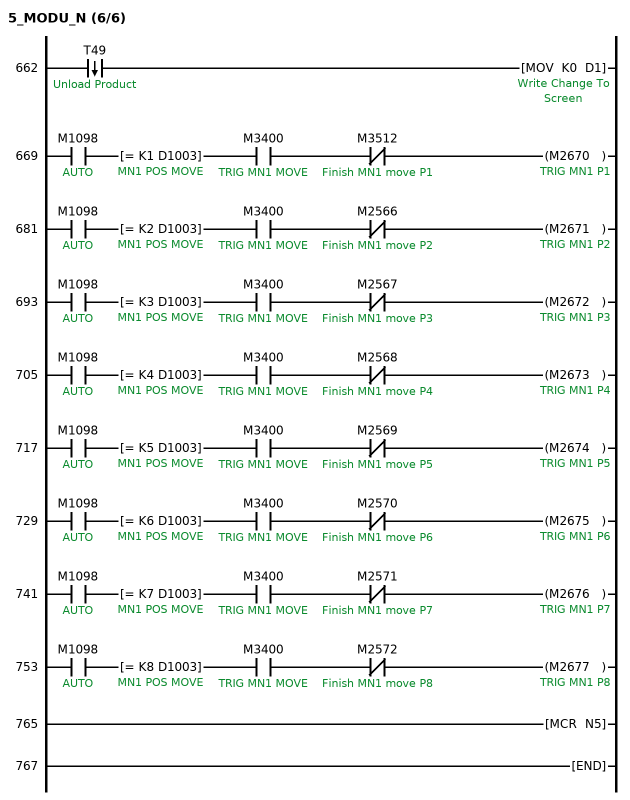
662   LDF     T49  ; Unload Product
      MOV     K0 D1
669   LD      M1098  ; AUTO
      AND=    K1 D1003  ; MN1 POS MOVE
      AND     M3400  ; TRIG MN1 MOVE
      ANI     M3512  ; Finish MN1 move P1
      OUT     M2670  ; TRIG MN1 P1
681   LD      M1098  ; AUTO
      AND=    K2 D1003  ; MN1 POS MOVE
      AND     M3400  ; TRIG MN1 MOVE
      ANI     M2566  ; Finish MN1 move P2
      OUT     M2671  ; TRIG MN1 P2
693   LD      M1098  ; AUTO
      AND=    K3 D1003  ; MN1 POS MOVE
      AND     M3400  ; TRIG MN1 MOVE
      ANI     M2567  ; Finish MN1 move P3
      OUT     M2672  ; TRIG MN1 P3
705   LD      M1098  ; AUTO
      AND=    K4 D1003  ; MN1 POS MOVE
      AND     M3400  ; TRIG MN1 MOVE
      ANI     M2568  ; Finish MN1 move P4
      OUT     M2673  ; TRIG MN1 P4
717   LD      M1098  ; AUTO
      AND=    K5 D1003  ; MN1 POS MOVE
      AND     M3400  ; TRIG MN1 MOVE
      ANI     M2569  ; Finish MN1 move P5
      OUT     M2674  ; TRIG MN1 P5
729   LD      M1098  ; AUTO
      AND=    K6 D1003  ; MN1 POS MOVE
      AND     M3400  ; TRIG MN1 MOVE
      ANI     M2570  ; Finish MN1 move P6
      OUT     M2675  ; TRIG MN1 P6
741   LD      M1098  ; AUTO
      AND=    K7 D1003  ; MN1 POS MOVE
      AND     M3400  ; TRIG MN1 MOVE
      ANI     M2571  ; Finish MN1 move P7
      OUT     M2676  ; TRIG MN1 P7
753   LD      M1098  ; AUTO
      AND=    K8 D1003  ; MN1 POS MOVE
      AND     M3400  ; TRIG MN1 MOVE
      ANI     M2572  ; Finish MN1 move P8
      OUT     M2677  ; TRIG MN1 P8
765   MCR     N5
767   END
END_PROGRAM

PROGRAM 6_IO
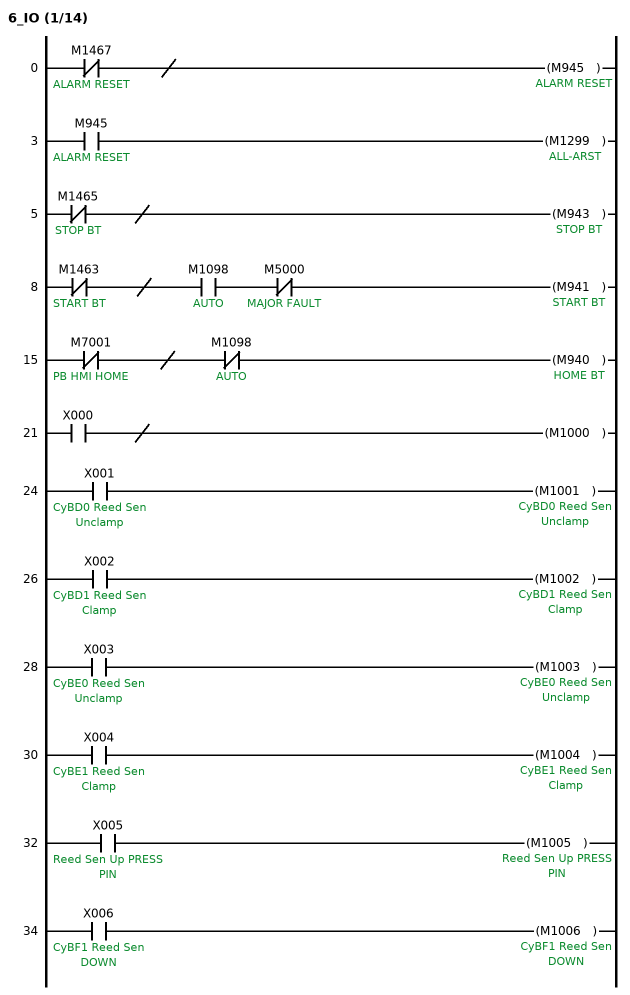
0     LDI     M1467  ; ALARM RESET
      INV
      OUT     M945  ; ALARM RESET
3     LD      M945  ; ALARM RESET
      OUT     M1299  ; ALL-ARST
5     LDI     M1465  ; STOP BT
      INV
      OUT     M943  ; STOP BT
8     LDI     M1463  ; START BT
      INV
      AND     M1098  ; AUTO
      ANI     M5000  ; MAJOR FAULT
      OUT     M941  ; START BT
15    LDI     M7001  ; PB HMI HOME
      INV
      ANI     M1098  ; AUTO
      OUT     M940  ; HOME BT
21    LD      X000
      INV
      OUT     M1000
24    LD      X001  ; CyBD0 Reed Sen Unclamp
      OUT     M1001  ; CyBD0 Reed Sen Unclamp
26    LD      X002  ; CyBD1 Reed Sen Clamp
      OUT     M1002  ; CyBD1 Reed Sen Clamp
28    LD      X003  ; CyBE0 Reed Sen Unclamp
      OUT     M1003  ; CyBE0 Reed Sen Unclamp
30    LD      X004  ; CyBE1 Reed Sen Clamp
      OUT     M1004  ; CyBE1 Reed Sen Clamp
32    LD      X005  ; Reed Sen Up PRESS PIN
      OUT     M1005  ; Reed Sen Up PRESS PIN
34    LD      X006  ; CyBF1 Reed Sen DOWN
      OUT     M1006  ; CyBF1 Reed Sen DOWN
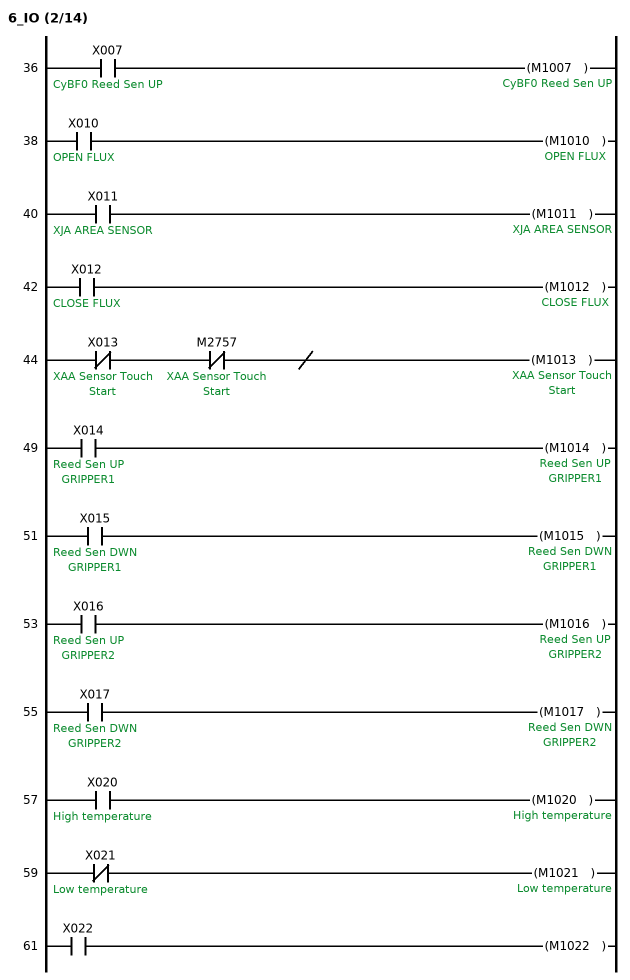
36    LD      X007  ; CyBF0 Reed Sen UP
      OUT     M1007  ; CyBF0 Reed Sen UP
38    LD      X010  ; OPEN FLUX
      OUT     M1010  ; OPEN FLUX
40    LD      X011  ; XJA AREA SENSOR
      OUT     M1011  ; XJA AREA SENSOR
42    LD      X012  ; CLOSE FLUX
      OUT     M1012  ; CLOSE FLUX
44    LDI     X013  ; XAA Sensor Touch Start
      ANI     M2757  ; XAA Sensor Touch Start
      INV
      OUT     M1013  ; XAA Sensor Touch Start
49    LD      X014  ; Reed Sen UP GRIPPER1
      OUT     M1014  ; Reed Sen UP GRIPPER1
51    LD      X015  ; Reed Sen DWN GRIPPER1
      OUT     M1015  ; Reed Sen DWN GRIPPER1
53    LD      X016  ; Reed Sen UP GRIPPER2
      OUT     M1016  ; Reed Sen UP GRIPPER2
55    LD      X017  ; Reed Sen DWN GRIPPER2
      OUT     M1017  ; Reed Sen DWN GRIPPER2
57    LD      X020  ; High temperature
      OUT     M1020  ; High temperature
59    LDI     X021  ; Low temperature
      OUT     M1021  ; Low temperature
61    LD      X022
      OUT     M1022
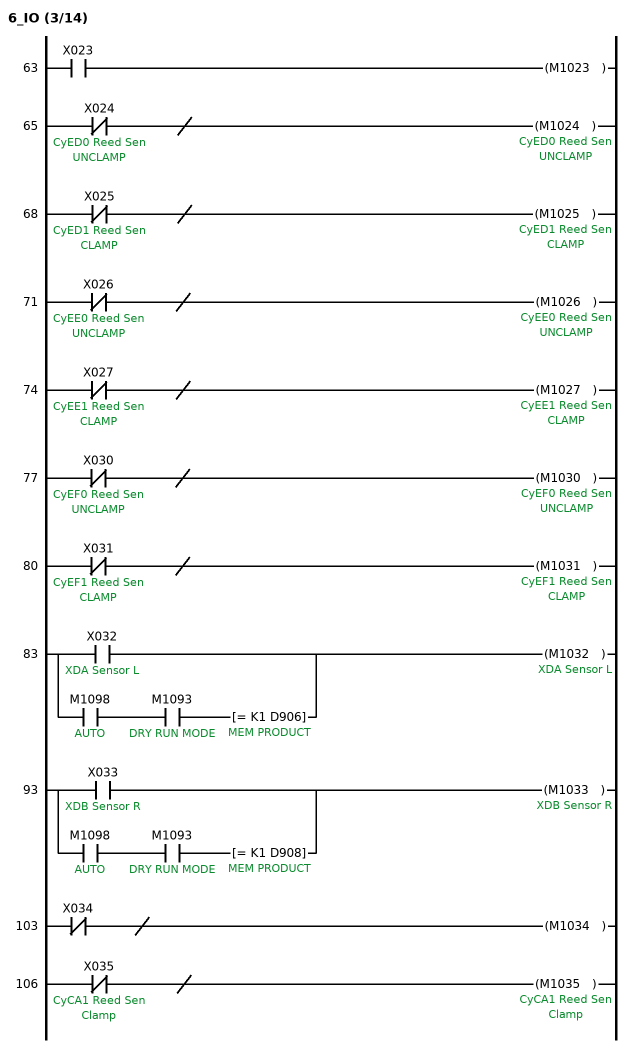
63    LD      X023
      OUT     M1023
65    LDI     X024  ; CyED0 Reed Sen UNCLAMP
      INV
      OUT     M1024  ; CyED0 Reed Sen UNCLAMP
68    LDI     X025  ; CyED1 Reed Sen CLAMP
      INV
      OUT     M1025  ; CyED1 Reed Sen CLAMP
71    LDI     X026  ; CyEE0 Reed Sen UNCLAMP
      INV
      OUT     M1026  ; CyEE0 Reed Sen UNCLAMP
74    LDI     X027  ; CyEE1 Reed Sen CLAMP
      INV
      OUT     M1027  ; CyEE1 Reed Sen CLAMP
77    LDI     X030  ; CyEF0 Reed Sen UNCLAMP
      INV
      OUT     M1030  ; CyEF0 Reed Sen UNCLAMP
80    LDI     X031  ; CyEF1 Reed Sen CLAMP
      INV
      OUT     M1031  ; CyEF1 Reed Sen CLAMP
83    LD      X032  ; XDA Sensor L
      LD      M1098  ; AUTO
      AND     M1093  ; DRY RUN MODE
      AND=    K1 D906  ; MEM PRODUCT
      ORB
      OUT     M1032  ; XDA Sensor L
93    LD      X033  ; XDB Sensor R
      LD      M1098  ; AUTO
      AND     M1093  ; DRY RUN MODE
      AND=    K1 D908  ; MEM PRODUCT
      ORB
      OUT     M1033  ; XDB Sensor R
103   LDI     X034
      INV
      OUT     M1034
106   LDI     X035  ; CyCA1 Reed Sen  Clamp
      INV
      OUT     M1035  ; CyCA1 Reed Sen  Clamp
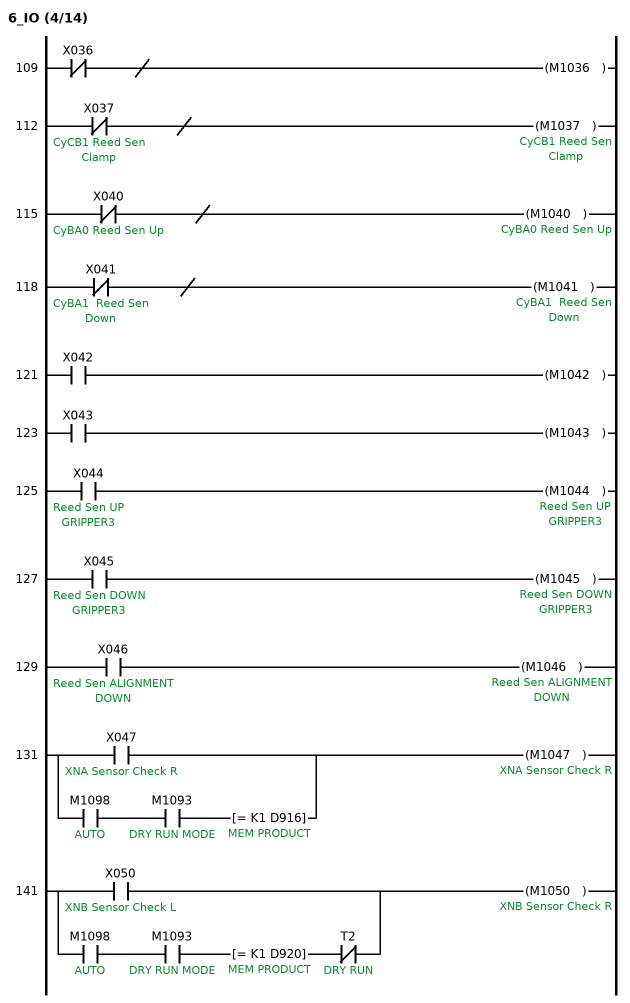
109   LDI     X036
      INV
      OUT     M1036
112   LDI     X037  ; CyCB1 Reed Sen  Clamp
      INV
      OUT     M1037  ; CyCB1 Reed Sen  Clamp
115   LDI     X040  ; CyBA0 Reed Sen Up
      INV
      OUT     M1040  ; CyBA0 Reed Sen Up
118   LDI     X041  ; CyBA1  Reed Sen Down
      INV
      OUT     M1041  ; CyBA1  Reed Sen Down
121   LD      X042
      OUT     M1042
123   LD      X043
      OUT     M1043
125   LD      X044  ; Reed Sen UP GRIPPER3
      OUT     M1044  ; Reed Sen UP GRIPPER3
127   LD      X045  ; Reed Sen DOWN GRIPPER3
      OUT     M1045  ; Reed Sen DOWN GRIPPER3
129   LD      X046  ; Reed Sen ALIGNMENT DOWN
      OUT     M1046  ; Reed Sen ALIGNMENT DOWN
131   LD      X047  ; XNA Sensor Check R
      LD      M1098  ; AUTO
      AND     M1093  ; DRY RUN MODE
      AND=    K1 D916  ; MEM PRODUCT
      ORB
      OUT     M1047  ; XNA Sensor Check R
141   LD      X050  ; XNB Sensor Check L
      LD      M1098  ; AUTO
      AND     M1093  ; DRY RUN MODE
      AND=    K1 D920  ; MEM PRODUCT
      ANI     T2  ; DRY RUN
      ORB
      OUT     M1050  ; XNB Sensor Check R
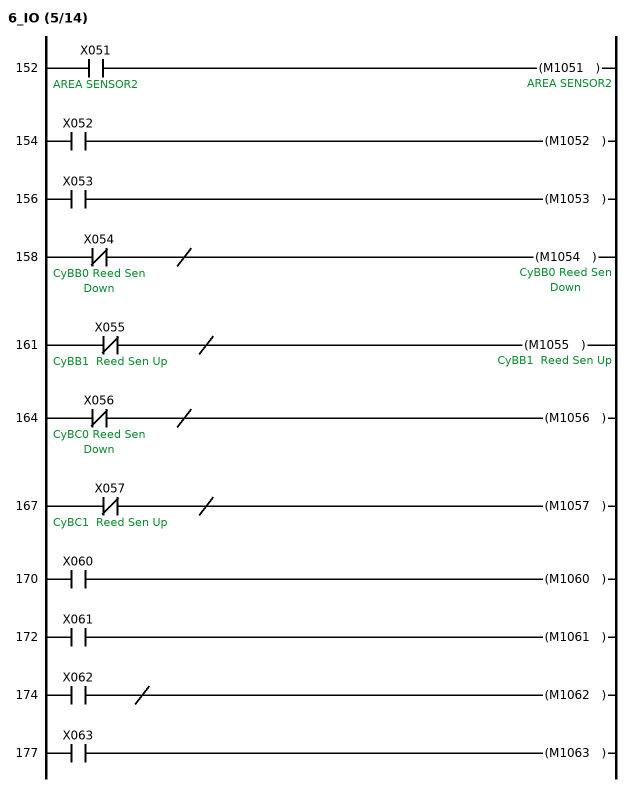
152   LD      X051  ; AREA SENSOR2
      OUT     M1051  ; AREA SENSOR2
154   LD      X052
      OUT     M1052
156   LD      X053
      OUT     M1053
158   LDI     X054  ; CyBB0 Reed Sen Down
      INV
      OUT     M1054  ; CyBB0 Reed Sen Down
161   LDI     X055  ; CyBB1  Reed Sen Up
      INV
      OUT     M1055  ; CyBB1  Reed Sen Up
164   LDI     X056  ; CyBC0 Reed Sen Down
      INV
      OUT     M1056
167   LDI     X057  ; CyBC1  Reed Sen Up
      INV
      OUT     M1057
170   LD      X060
      OUT     M1060
172   LD      X061
      OUT     M1061
174   LD      X062
      INV
      OUT     M1062
177   LD      X063
      OUT     M1063
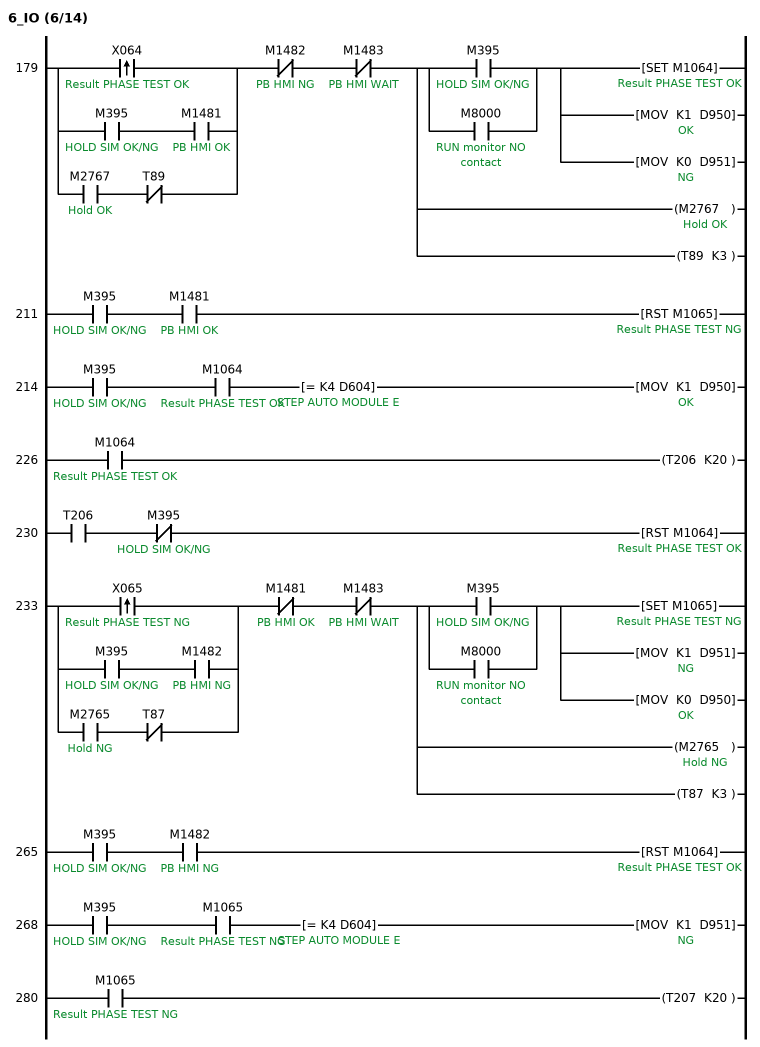
179   LDP     X064  ; Result PHASE TEST OK
      LD      M395  ; HOLD SIM OK/NG
      AND     M1481  ; PB HMI OK
      ORB
      LD      M2767  ; Hold OK
      ANI     T89
      ORB
      ANI     M1482  ; PB HMI NG
      ANI     M1483  ; PB HMI WAIT
      MPS
      LD      M395  ; HOLD SIM OK/NG
      OR      M8000  ; RUN monitor NO contact
      ANB
      SET     M1064  ; Result PHASE TEST OK
      MOV     K1 D950  ; OK
      MOV     K0 D951  ; NG
      MPP
      OUT     M2767  ; Hold OK
      OUT     T89 K3
211   LD      M395  ; HOLD SIM OK/NG
      AND     M1481  ; PB HMI OK
      RST     M1065  ; Result PHASE TEST NG
214   LD      M395  ; HOLD SIM OK/NG
      AND     M1064  ; Result PHASE TEST OK
      AND=    K4 D604  ; STEP AUTO MODULE E
      MOV     K1 D950
226   LD      M1064  ; Result PHASE TEST OK
      OUT     T206 K20
230   LD      T206
      ANI     M395  ; HOLD SIM OK/NG
      RST     M1064  ; Result PHASE TEST OK
233   LDP     X065  ; Result PHASE TEST NG
      LD      M395  ; HOLD SIM OK/NG
      AND     M1482  ; PB HMI NG
      ORB
      LD      M2765  ; Hold NG
      ANI     T87
      ORB
      ANI     M1481  ; PB HMI OK
      ANI     M1483  ; PB HMI WAIT
      MPS
      LD      M395  ; HOLD SIM OK/NG
      OR      M8000  ; RUN monitor NO contact
      ANB
      SET     M1065  ; Result PHASE TEST NG
      MOV     K1 D951
      MOV     K0 D950
      MPP
      OUT     M2765  ; Hold NG
      OUT     T87 K3
265   LD      M395  ; HOLD SIM OK/NG
      AND     M1482  ; PB HMI NG
      RST     M1064  ; Result PHASE TEST OK
268   LD      M395  ; HOLD SIM OK/NG
      AND     M1065  ; Result PHASE TEST NG
      AND=    K4 D604  ; STEP AUTO MODULE E
      MOV     K1 D951
280   LD      M1065  ; Result PHASE TEST NG
      OUT     T207 K20
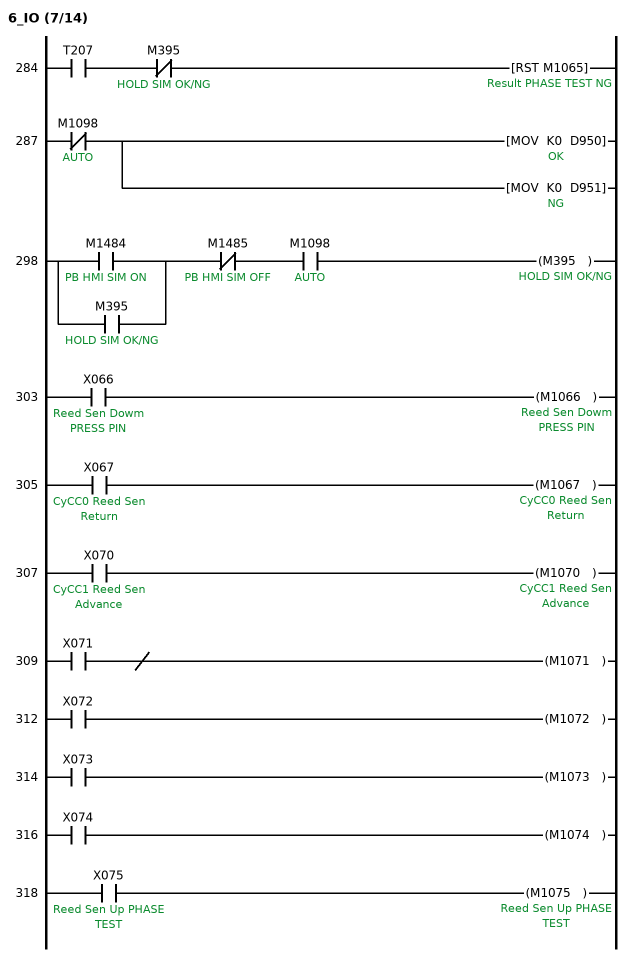
284   LD      T207
      ANI     M395  ; HOLD SIM OK/NG
      RST     M1065  ; Result PHASE TEST NG
287   LDI     M1098  ; AUTO
      MOV     K0 D950
      MOV     K0 D951
298   LD      M1484  ; PB HMI SIM ON
      OR      M395  ; HOLD SIM OK/NG
      ANI     M1485  ; PB HMI SIM OFF
      AND     M1098  ; AUTO
      OUT     M395  ; HOLD SIM OK/NG
303   LD      X066  ; Reed Sen Dowm PRESS PIN
      OUT     M1066  ; Reed Sen Dowm PRESS PIN
305   LD      X067  ; CyCC0 Reed Sen Return
      OUT     M1067  ; CyCC0 Reed Sen Return
307   LD      X070  ; CyCC1 Reed Sen  Advance
      OUT     M1070  ; CyCC1 Reed Sen  Advance
309   LD      X071
      INV
      OUT     M1071
312   LD      X072
      OUT     M1072
314   LD      X073
      OUT     M1073
316   LD      X074
      OUT     M1074
318   LD      X075  ; Reed Sen Up PHASE TEST
      OUT     M1075  ; Reed Sen Up PHASE TEST
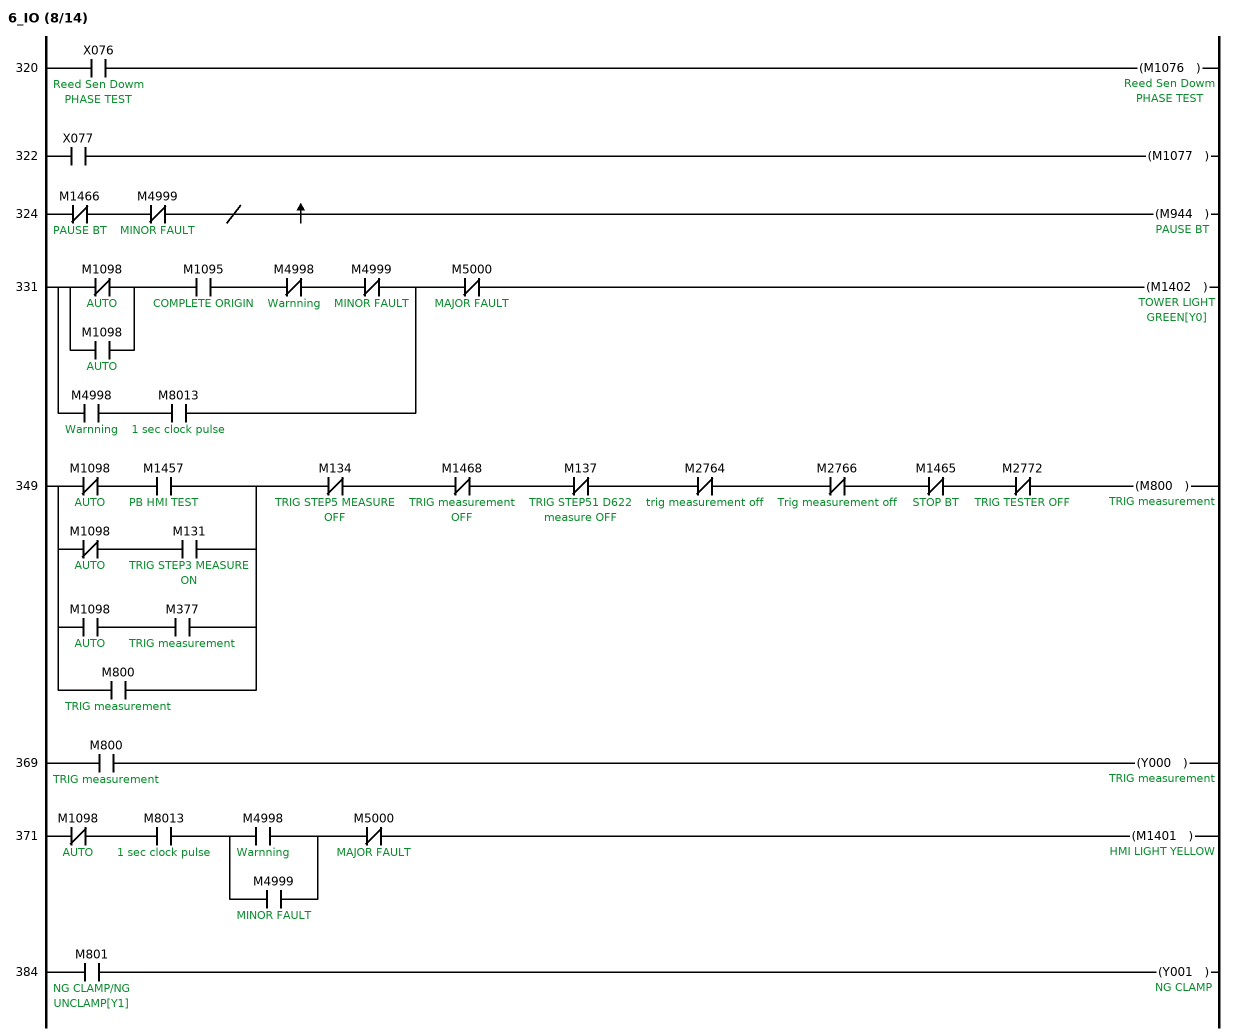
320   LD      X076  ; Reed Sen Dowm PHASE TEST
      OUT     M1076  ; Reed Sen Dowm PHASE TEST
322   LD      X077
      OUT     M1077
324   LDI     M1466  ; PAUSE BT
      ANI     M4999  ; MINOR FAULT
      INV
      MEP
      OUT     M944  ; PAUSE BT
331   LDI     M1098  ; AUTO
      OR      M1098  ; AUTO
      AND     M1095  ; COMPLETE ORIGIN
      ANI     M4998  ; Warnning
      ANI     M4999  ; MINOR FAULT
      LD      M4998  ; Warnning
      AND     M8013  ; 1 sec clock pulse
      ORB
      ANI     M5000  ; MAJOR FAULT
      OUT     M1402  ; TOWER LIGHT GREEN[Y0]
349   LDI     M1098  ; AUTO
      AND     M1457  ; PB HMI TEST
      LDI     M1098  ; AUTO
      AND     M131  ; TRIG STEP3 MEASURE ON
      ORB
      LD      M1098  ; AUTO
      AND     M377  ; TRIG measurement
      ORB
      OR      M800  ; TRIG measurement
      ANI     M134  ; TRIG STEP5 MEASURE OFF
      ANI     M1468  ; TRIG measurement OFF
      ANI     M137  ; TRIG STEP51 D622 measure OFF
      ANI     M2764  ; trig measurement off
      ANI     M2766  ; Trig measurement off
      ANI     M1465  ; STOP BT
      ANI     M2772  ; TRIG TESTER OFF
      OUT     M800  ; TRIG measurement
369   LD      M800  ; TRIG measurement
      OUT     Y000  ; TRIG measurement
371   LDI     M1098  ; AUTO
      AND     M8013  ; 1 sec clock pulse
      LD      M4998  ; Warnning
      OR      M4999  ; MINOR FAULT
      ANB
      ANI     M5000  ; MAJOR FAULT
      OUT     M1401  ; HMI LIGHT YELLOW
384   LD      M801  ; NG CLAMP/NG UNCLAMP[Y1]
      OUT     Y001  ; NG CLAMP
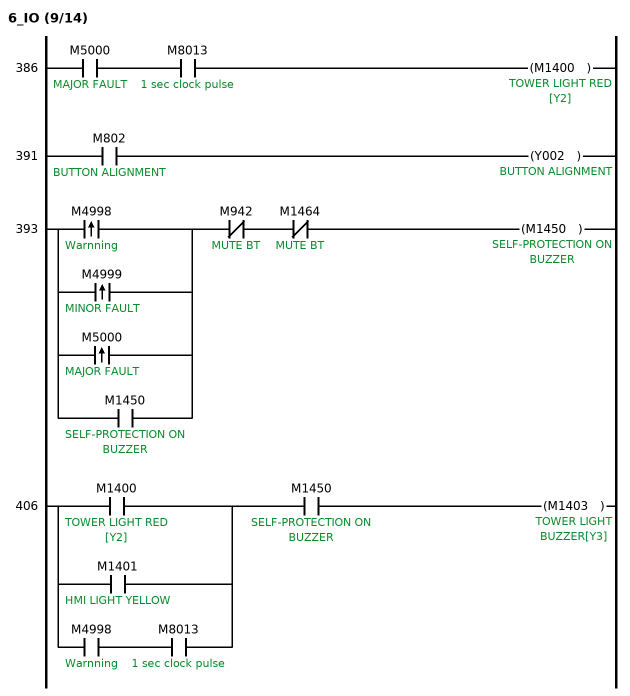
386   LD      M5000  ; MAJOR FAULT
      AND     M8013  ; 1 sec clock pulse
      OUT     M1400  ; TOWER LIGHT RED [Y2]
391   LD      M802  ; BUTTON ALIGNMENT
      OUT     Y002  ; BUTTON ALIGNMENT
393   LDP     M4998  ; Warnning
      ORP     M4999  ; MINOR FAULT
      ORP     M5000  ; MAJOR FAULT
      OR      M1450  ; SELF-PROTECTION ON BUZZER
      ANI     M942  ; MUTE BT
      ANI     M1464  ; MUTE BT
      OUT     M1450  ; SELF-PROTECTION ON BUZZER
406   LD      M1400  ; TOWER LIGHT RED [Y2]
      OR      M1401  ; HMI LIGHT YELLOW
      LD      M4998  ; Warnning
      AND     M8013  ; 1 sec clock pulse
      ORB
      AND     M1450  ; SELF-PROTECTION ON BUZZER
      OUT     M1403  ; TOWER LIGHT BUZZER[Y3]
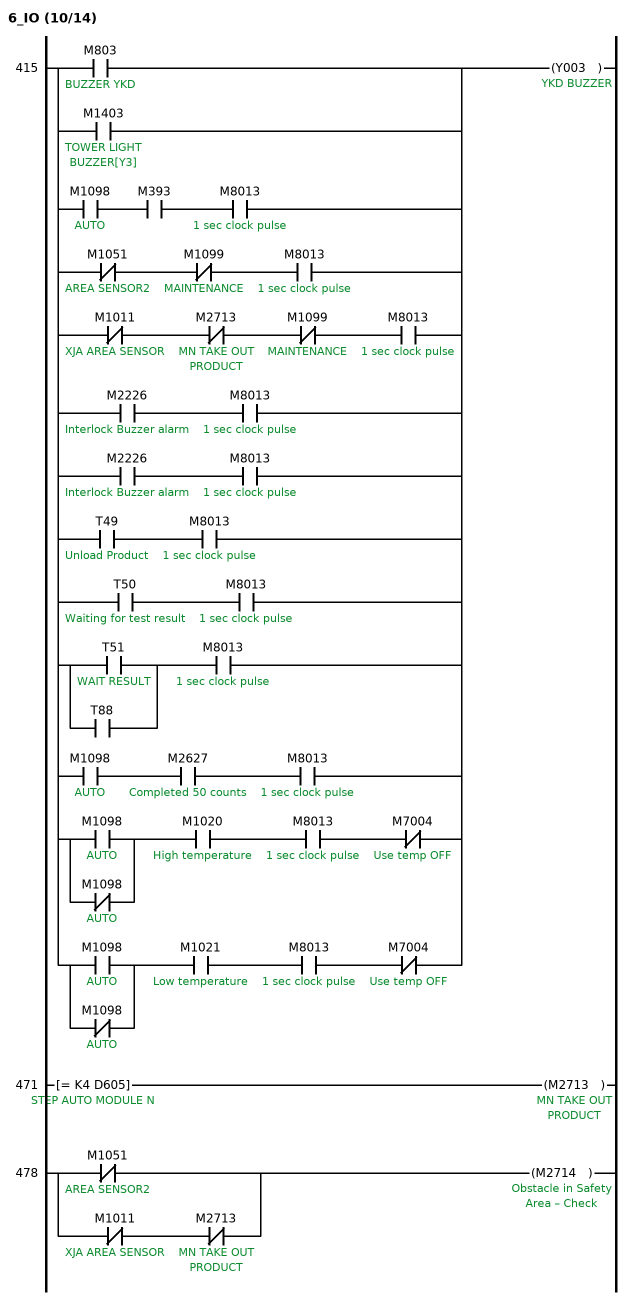
415   LD      M803  ; BUZZER YKD
      OR      M1403  ; TOWER LIGHT BUZZER[Y3]
      LD      M1098  ; AUTO
      AND     M393
      AND     M8013  ; 1 sec clock pulse
      ORB
      LDI     M1051  ; AREA SENSOR2
      ANI     M1099  ; MAINTENANCE
      AND     M8013  ; 1 sec clock pulse
      ORB
      LDI     M1011  ; XJA AREA SENSOR
      ANI     M2713  ; MN TAKE OUT PRODUCT
      ANI     M1099  ; MAINTENANCE
      AND     M8013  ; 1 sec clock pulse
      ORB
      LD      M2226  ; Interlock Buzzer alarm
      AND     M8013  ; 1 sec clock pulse
      ORB
      LD      M2226  ; Interlock Buzzer alarm
      AND     M8013  ; 1 sec clock pulse
      ORB
      LD      T49  ; Unload Product
      AND     M8013  ; 1 sec clock pulse
      ORB
      LD      T50  ; Waiting for test result
      AND     M8013  ; 1 sec clock pulse
      ORB
      LD      T51  ; WAIT RESULT
      OR      T88
      AND     M8013  ; 1 sec clock pulse
      ORB
      LD      M1098  ; AUTO
      AND     M2627  ; Completed 50 counts
      AND     M8013  ; 1 sec clock pulse
      ORB
      LD      M1098  ; AUTO
      ORI     M1098  ; AUTO
      AND     M1020  ; High temperature
      AND     M8013  ; 1 sec clock pulse
      ANI     M7004  ; Use temp OFF
      ORB
      LD      M1098  ; AUTO
      ORI     M1098  ; AUTO
      AND     M1021  ; Low temperature
      AND     M8013  ; 1 sec clock pulse
      ANI     M7004  ; Use temp OFF
      ORB
      OUT     Y003  ; YKD BUZZER
471   LD=     K4 D605  ; STEP AUTO MODULE N
      OUT     M2713  ; MN TAKE OUT PRODUCT
478   LDI     M1051  ; AREA SENSOR2
      LDI     M1011  ; XJA AREA SENSOR
      ANI     M2713  ; MN TAKE OUT PRODUCT
      ORB
      OUT     M2714  ; Obstacle in Safety Area – Check
